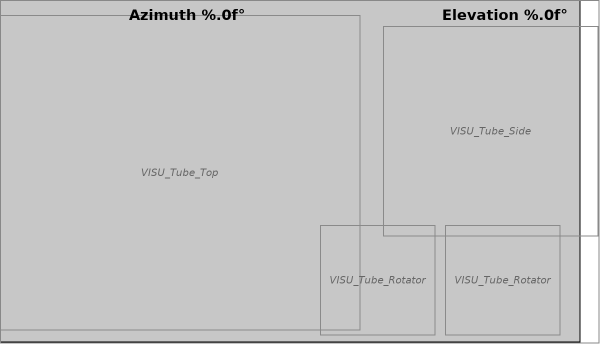
VISUALIZATION VISU_AxesImage  // 600x344
VAR_IN_OUT
	ref : Axes;
    widget : AxesWidget;
END_VAR
    Rectangle (0,0 580x342)
    Frame (383,26 215x210)
        shows VISU_Tube_Side(ele := widget.image.ele, eleTarget := widget.image.eleTarget, eleTargetInvisible := widget.image.eleTargetInvisible, mark10Degrees := widget.image.mark10Degrees)
    Frame (0,15 360x315)
        shows VISU_Tube_Top(widget := widget.image)
    Rectangle (90,5 195x20), "Azimuth %.0f°", text variable: ref.feedback.aziPos.degrees.value
    Rectangle (435,5 140x20), "Elevation %.0f°", text variable: ref.feedback.elePos.degrees.value
    Frame (320,225 115x110)
        shows VISU_Tube_Rotator(stationName := widget.image.rocStationName, name := widget.image.rocName, rotAngle := widget.image.roc)
    Frame (445,225 115x110)
        shows VISU_Tube_Rotator(stationName := widget.image.ronStationName, name := widget.image.ronName, rotAngle := widget.image.ron)
END_VISUALIZATION

(* stored: Version 1.1.0.1, ProductVersion 3.1.4019.2
   Visu VISU_AxesImage: Id {71248f03-e3a3-4692-a591-002b8c7e899b} *)
